# EPICS autosave request: softGlueApp/Db/MCSAsub_settings.req
$(P)$(Q)MCS.A
$(P)$(Q)MCS.E
